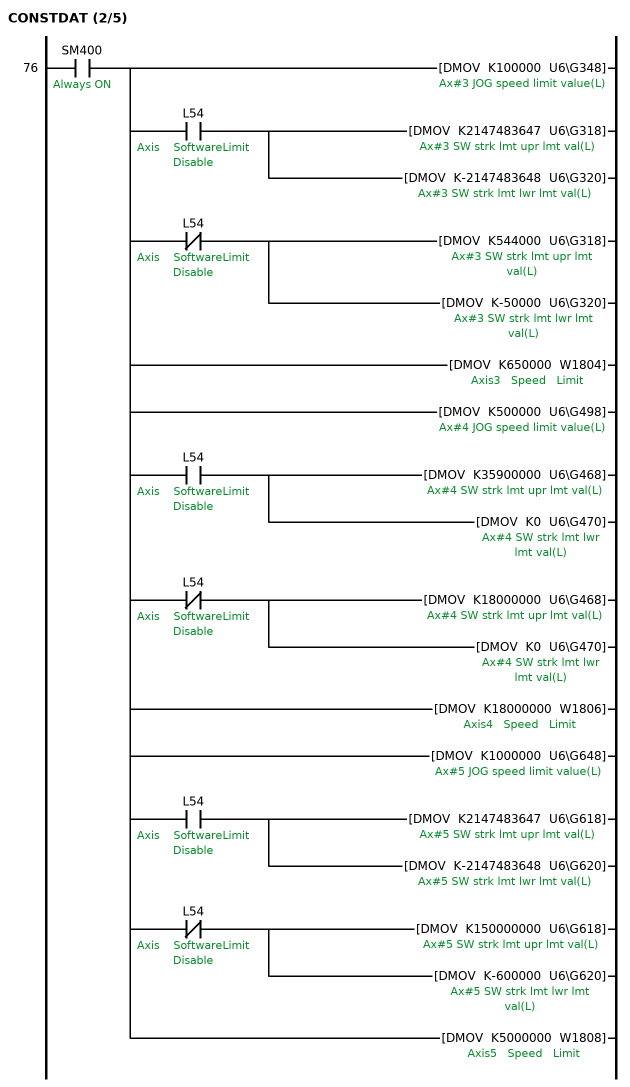
[picture p48: ladder of CONSTDAT, rungs at steps 76 to 76]
76    LD      SM400  ; Always ON
      DMOV    K100000 U6\G348  ; Ax#3 JOG speed limit value(L)
      MPS
      AND     L54  ; Axis    SoftwareLimit   Disable
      DMOV    K2147483647 U6\G318  ; Ax#3 SW strk lmt upr lmt val(L)
      DMOV    K-2147483648 U6\G320  ; Ax#3 SW strk lmt lwr lmt val(L)
      MRD
      ANI     L54  ; Axis    SoftwareLimit   Disable
      DMOV    K544000 U6\G318
      DMOV    K-50000 U6\G320
      MPP
      DMOV    K650000 W1804  ; Axis3   Speed   Limit
      DMOV    K500000 U6\G498  ; Ax#4 JOG speed limit value(L)
      MPS
      AND     L54  ; Axis    SoftwareLimit   Disable
      DMOV    K35900000 U6\G468  ; Ax#4 SW strk lmt upr lmt val(L)
      DMOV    K0 U6\G470  ; Ax#4 SW strk lmt lwr lmt val(L)
      MRD
      ANI     L54  ; Axis    SoftwareLimit   Disable
      DMOV    K18000000 U6\G468
      DMOV    K0 U6\G470
      MPP
      DMOV    K18000000 W1806  ; Axis4   Speed   Limit
      DMOV    K1000000 U6\G648  ; Ax#5 JOG speed limit value(L)
      MPS
      AND     L54  ; Axis    SoftwareLimit   Disable
      DMOV    K2147483647 U6\G618  ; Ax#5 SW strk lmt upr lmt val(L)
      DMOV    K-2147483648 U6\G620  ; Ax#5 SW strk lmt lwr lmt val(L)
      MRD
      ANI     L54  ; Axis    SoftwareLimit   Disable
      DMOV    K150000000 U6\G618
      DMOV    K-600000 U6\G620
      MPP
      DMOV    K5000000 W1808  ; Axis5   Speed   Limit
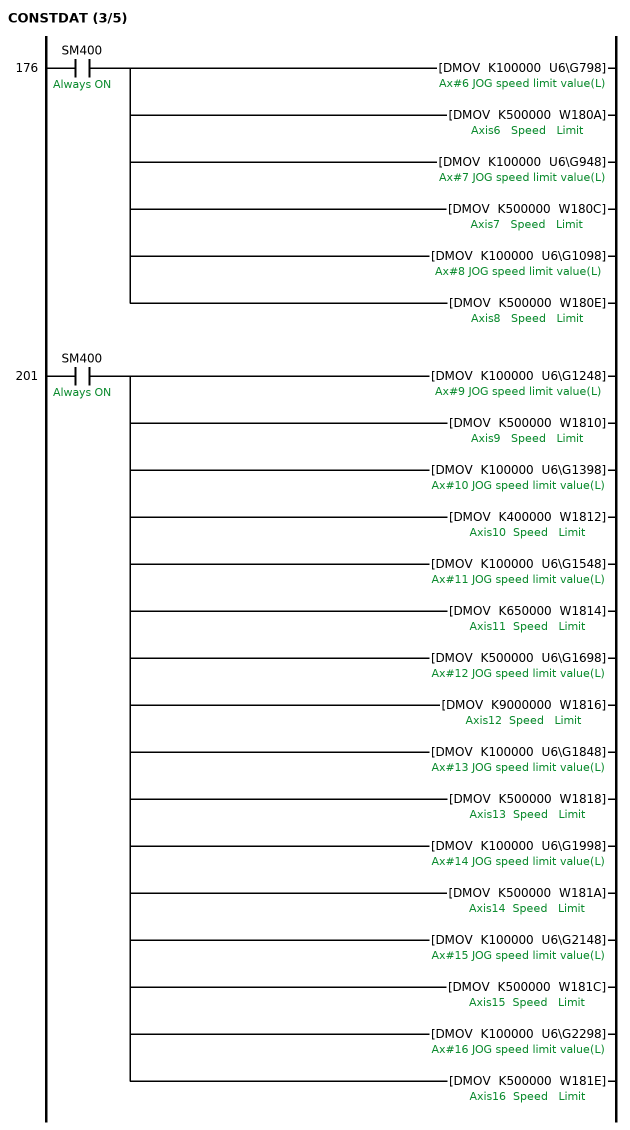
176   LD      SM400  ; Always ON
      DMOV    K100000 U6\G798  ; Ax#6 JOG speed limit value(L)
      DMOV    K500000 W180A  ; Axis6   Speed   Limit
      DMOV    K100000 U6\G948  ; Ax#7 JOG speed limit value(L)
      DMOV    K500000 W180C  ; Axis7   Speed   Limit
      DMOV    K100000 U6\G1098  ; Ax#8 JOG speed limit value(L)
      DMOV    K500000 W180E  ; Axis8   Speed   Limit
201   LD      SM400  ; Always ON
      DMOV    K100000 U6\G1248  ; Ax#9 JOG speed limit value(L)
      DMOV    K500000 W1810  ; Axis9   Speed   Limit
      DMOV    K100000 U6\G1398  ; Ax#10 JOG speed limit value(L)
      DMOV    K400000 W1812  ; Axis10  Speed   Limit
      DMOV    K100000 U6\G1548  ; Ax#11 JOG speed limit value(L)
      DMOV    K650000 W1814  ; Axis11  Speed   Limit
      DMOV    K500000 U6\G1698  ; Ax#12 JOG speed limit value(L)
      DMOV    K9000000 W1816  ; Axis12  Speed   Limit
      DMOV    K100000 U6\G1848  ; Ax#13 JOG speed limit value(L)
      DMOV    K500000 W1818  ; Axis13  Speed   Limit
      DMOV    K100000 U6\G1998  ; Ax#14 JOG speed limit value(L)
      DMOV    K500000 W181A  ; Axis14  Speed   Limit
      DMOV    K100000 U6\G2148  ; Ax#15 JOG speed limit value(L)
      DMOV    K500000 W181C  ; Axis15  Speed   Limit
      DMOV    K100000 U6\G2298  ; Ax#16 JOG speed limit value(L)
      DMOV    K500000 W181E  ; Axis16  Speed   Limit
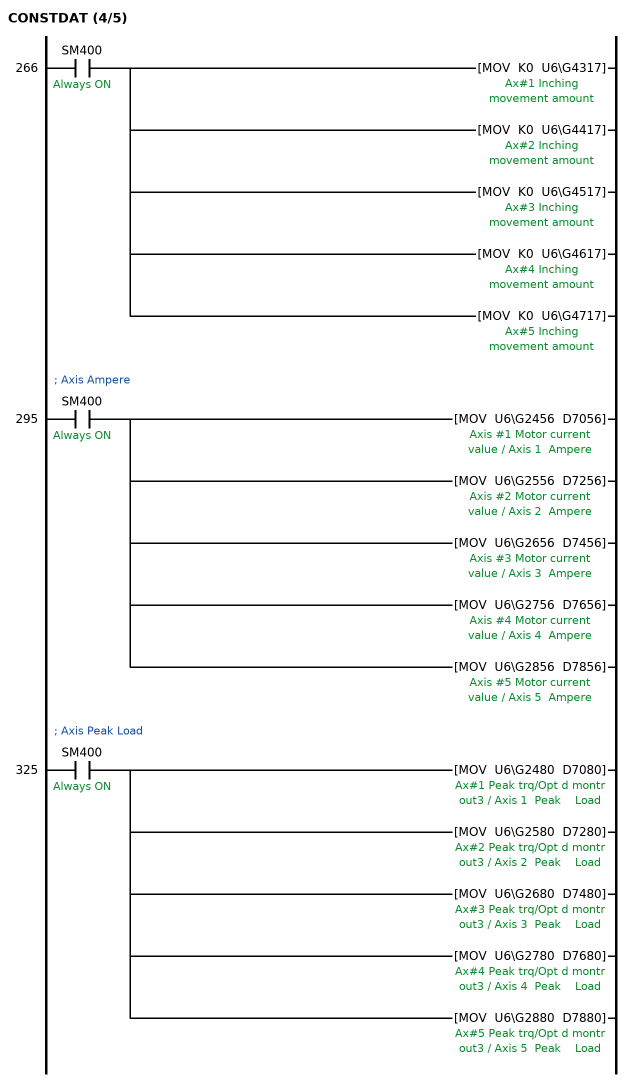
266   LD      SM400  ; Always ON
      MOV     K0 U6\G4317  ; Ax#1 Inching movement amount
      MOV     K0 U6\G4417  ; Ax#2 Inching movement amount
      MOV     K0 U6\G4517  ; Ax#3 Inching movement amount
      MOV     K0 U6\G4617  ; Ax#4 Inching movement amount
      MOV     K0 U6\G4717  ; Ax#5 Inching movement amount
; Axis Ampere
295   LD      SM400  ; Always ON
      MOV     U6\G2456 D7056  ; Axis #1 Motor current value / Axis 1  Ampere
      MOV     U6\G2556 D7256  ; Axis #2 Motor current value / Axis 2  Ampere
      MOV     U6\G2656 D7456  ; Axis #3 Motor current value / Axis 3  Ampere
      MOV     U6\G2756 D7656  ; Axis #4 Motor current value / Axis 4  Ampere
      MOV     U6\G2856 D7856  ; Axis #5 Motor current value / Axis 5  Ampere
; Axis Peak Load
325   LD      SM400  ; Always ON
      MOV     U6\G2480 D7080  ; Ax#1 Peak trq/Opt d montr out3 / Axis 1  Peak    Load
      MOV     U6\G2580 D7280  ; Ax#2 Peak trq/Opt d montr out3 / Axis 2  Peak    Load
      MOV     U6\G2680 D7480  ; Ax#3 Peak trq/Opt d montr out3 / Axis 3  Peak    Load
      MOV     U6\G2780 D7680  ; Ax#4 Peak trq/Opt d montr out3 / Axis 4  Peak    Load
      MOV     U6\G2880 D7880  ; Ax#5 Peak trq/Opt d montr out3 / Axis 5  Peak    Load
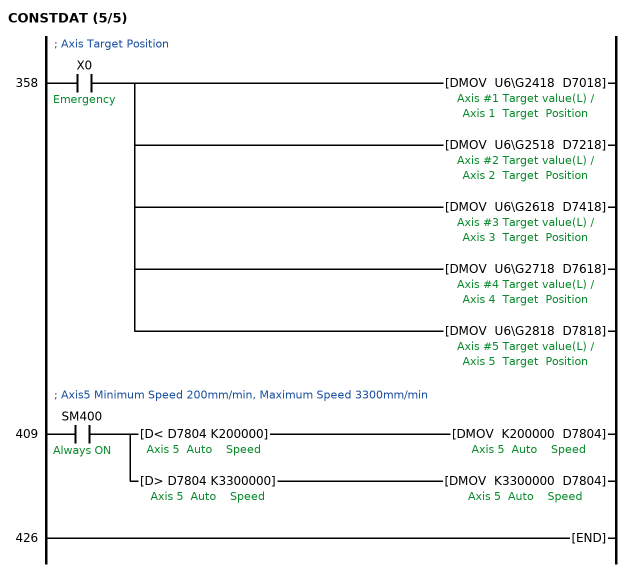
; Axis Target Position
358   LD      X0  ; Emergency
      DMOV    U6\G2418 D7018  ; Axis #1 Target value(L) / Axis 1  Target  Position
      DMOV    U6\G2518 D7218  ; Axis #2 Target value(L) / Axis 2  Target  Position
      DMOV    U6\G2618 D7418  ; Axis #3 Target value(L) / Axis 3  Target  Position
      DMOV    U6\G2718 D7618  ; Axis #4 Target value(L) / Axis 4  Target  Position
      DMOV    U6\G2818 D7818  ; Axis #5 Target value(L) / Axis 5  Target  Position
; Axis5 Minimum Speed 200mm/min, Maximum Speed 3300mm/min
409   LD      SM400  ; Always ON
      MPS
      ANDD<   D7804 K200000  ; Axis 5  Auto    Speed
      DMOV    K200000 D7804
      MPP
      ANDD>   D7804 K3300000  ; Axis 5  Auto    Speed
      DMOV    K3300000 D7804
426   END
END_PROGRAM

PROGRAM Y_OUT
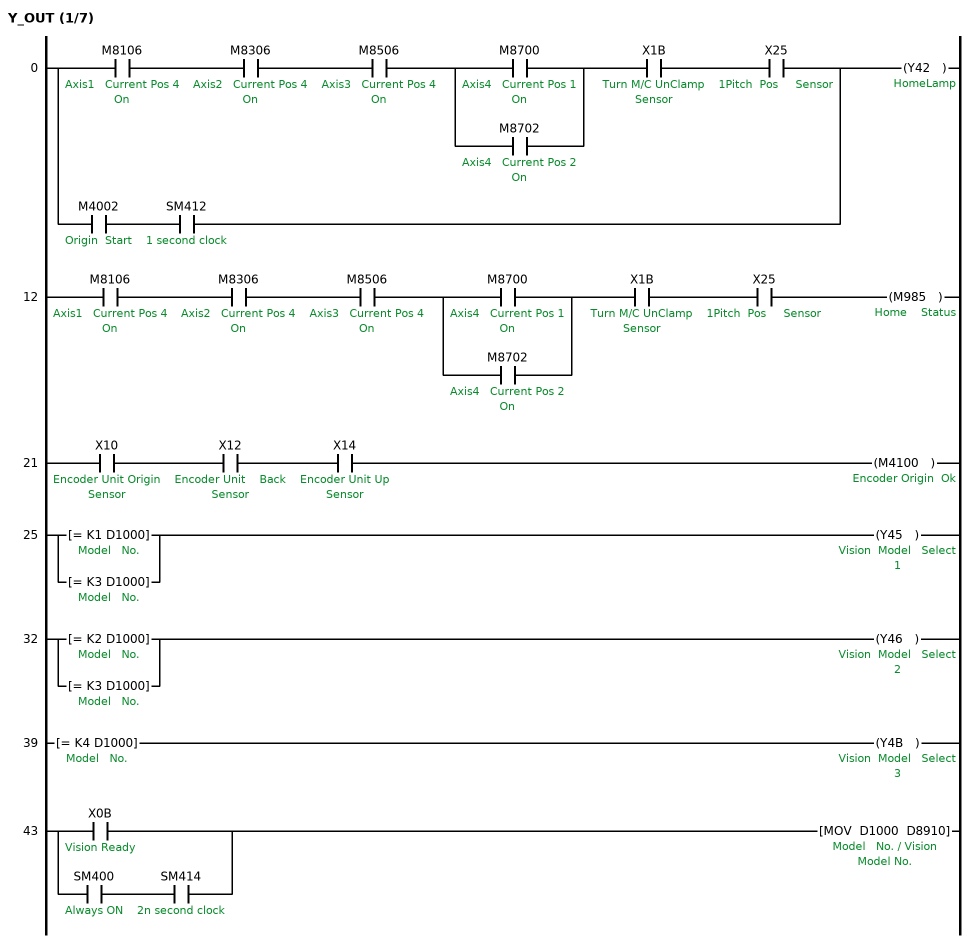
0     LD      M8106  ; Axis1   Current Pos 4 On
      AND     M8306  ; Axis2   Current Pos 4 On
      AND     M8506  ; Axis3   Current Pos 4 On
      LD      M8700  ; Axis4   Current Pos 1 On
      OR      M8702  ; Axis4   Current Pos 2 On
      ANB
      AND     X1B  ; Turn M/C UnClamp Sensor
      AND     X25  ; 1Pitch  Pos     Sensor
      LD      M4002  ; Origin  Start
      AND     SM412  ; 1 second clock
      ORB
      OUT     Y42  ; HomeLamp
12    LD      M8106  ; Axis1   Current Pos 4 On
      AND     M8306  ; Axis2   Current Pos 4 On
      AND     M8506  ; Axis3   Current Pos 4 On
      LD      M8700  ; Axis4   Current Pos 1 On
      OR      M8702  ; Axis4   Current Pos 2 On
      ANB
      AND     X1B  ; Turn M/C UnClamp Sensor
      AND     X25  ; 1Pitch  Pos     Sensor
      OUT     M985  ; Home    Status
21    LD      X10  ; Encoder Unit Origin Sensor
      AND     X12  ; Encoder Unit    Back    Sensor
      AND     X14  ; Encoder Unit Up Sensor
      OUT     M4100  ; Encoder Origin  Ok
25    LD=     K1 D1000  ; Model   No.
      OR=     K3 D1000  ; Model   No.
      OUT     Y45  ; Vision  Model   Select 1
32    LD=     K2 D1000  ; Model   No.
      OR=     K3 D1000  ; Model   No.
      OUT     Y46  ; Vision  Model   Select 2
39    LD=     K4 D1000  ; Model   No.
      OUT     Y4B  ; Vision  Model   Select 3
43    LD      X0B  ; Vision Ready
      LD      SM400  ; Always ON
      AND     SM414  ; 2n second clock
      ORB
      MOV     D1000 D8910  ; Vision Model No.
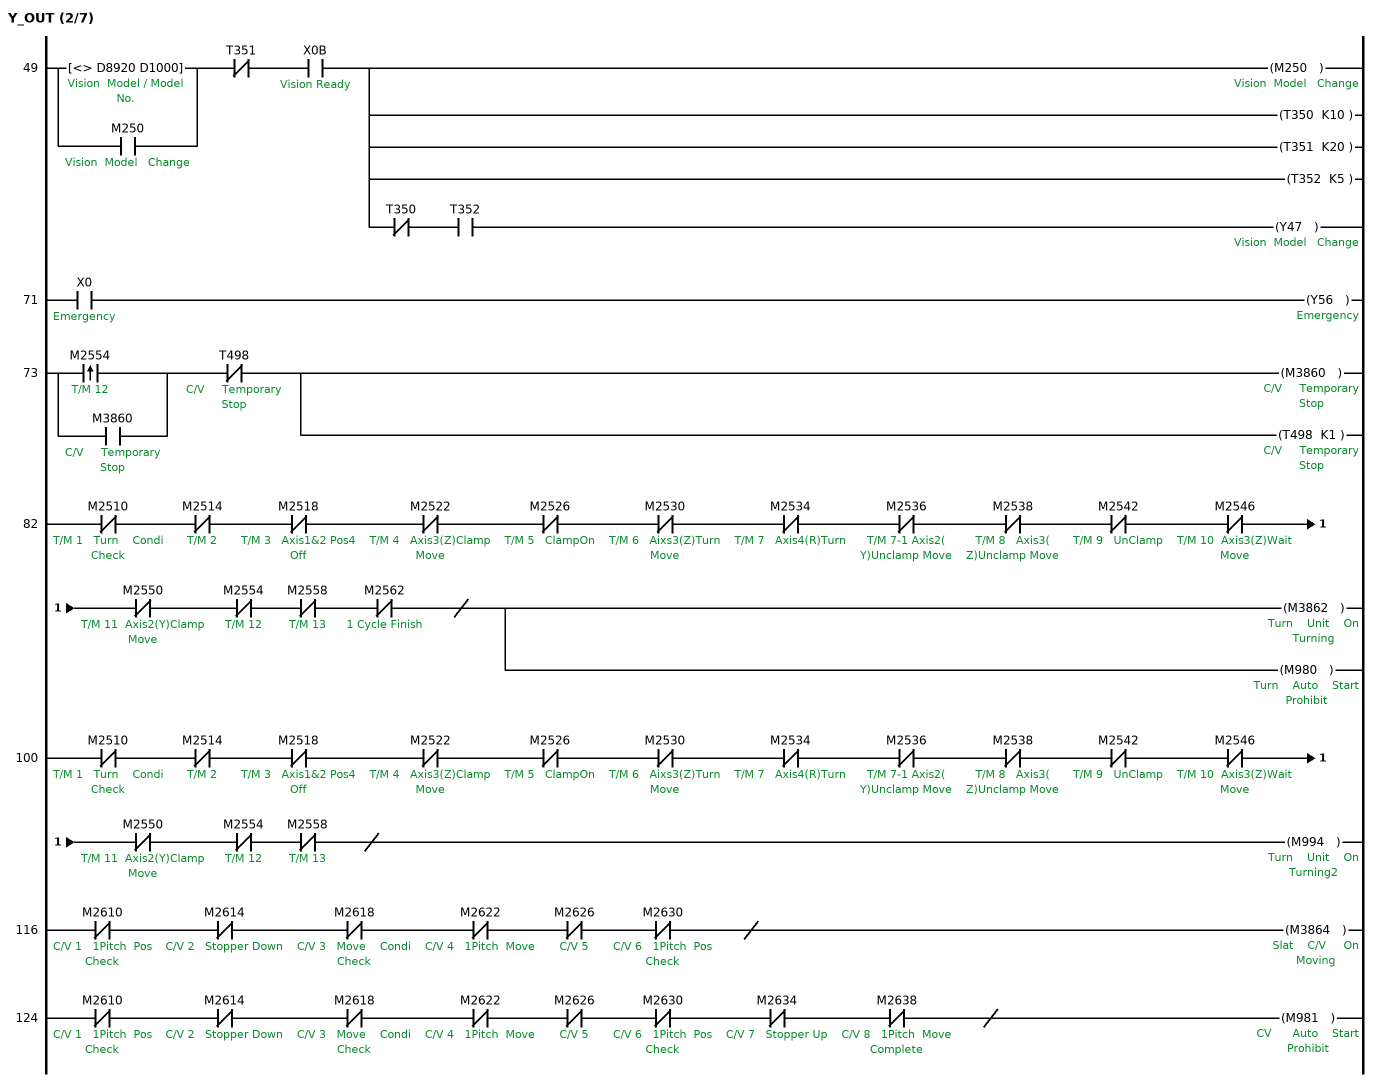
49    LD<>    D8920 D1000  ; Vision  Model / Model   No.
      OR      M250  ; Vision  Model   Change
      ANI     T351
      AND     X0B  ; Vision Ready
      OUT     M250  ; Vision  Model   Change
      OUT     T350 K10
      OUT     T351 K20
      OUT     T352 K5
      ANI     T350
      AND     T352
      OUT     Y47  ; Vision  Model   Change
71    LD      X0  ; Emergency
      OUT     Y56  ; Emergency
73    LDP     M2554  ; T/M 12
      OR      M3860  ; C/V     Temporary  Stop
      ANI     T498  ; C/V     Temporary  Stop
      OUT     M3860  ; C/V     Temporary  Stop
      OUT     T498 K1  ; C/V     Temporary  Stop
82    LDI     M2510  ; T/M 1   Turn    Condi   Check
      ANI     M2514  ; T/M 2
      ANI     M2518  ; T/M 3   Axis1&2 Pos4    Off
      ANI     M2522  ; T/M 4   Axis3(Z)Clamp   Move
      ANI     M2526  ; T/M 5   ClampOn
      ANI     M2530  ; T/M 6   Aixs3(Z)Turn    Move
      ANI     M2534  ; T/M 7   Axis4(R)Turn
      ANI     M2536  ; T/M 7-1 Axis2(Y)Unclamp Move
      ANI     M2538  ; T/M 8   Axis3(Z)Unclamp Move
      ANI     M2542  ; T/M 9   UnClamp
      ANI     M2546  ; T/M 10  Axis3(Z)Wait    Move
      ANI     M2550  ; T/M 11  Axis2(Y)Clamp   Move
      ANI     M2554  ; T/M 12
      ANI     M2558  ; T/M 13
      ANI     M2562  ; 1 Cycle Finish
      INV
      OUT     M3862  ; Turn    Unit    On      Turning
      OUT     M980  ; Turn    Auto    Start   Prohibit
100   LDI     M2510  ; T/M 1   Turn    Condi   Check
      ANI     M2514  ; T/M 2
      ANI     M2518  ; T/M 3   Axis1&2 Pos4    Off
      ANI     M2522  ; T/M 4   Axis3(Z)Clamp   Move
      ANI     M2526  ; T/M 5   ClampOn
      ANI     M2530  ; T/M 6   Aixs3(Z)Turn    Move
      ANI     M2534  ; T/M 7   Axis4(R)Turn
      ANI     M2536  ; T/M 7-1 Axis2(Y)Unclamp Move
      ANI     M2538  ; T/M 8   Axis3(Z)Unclamp Move
      ANI     M2542  ; T/M 9   UnClamp
      ANI     M2546  ; T/M 10  Axis3(Z)Wait    Move
      ANI     M2550  ; T/M 11  Axis2(Y)Clamp   Move
      ANI     M2554  ; T/M 12
      ANI     M2558  ; T/M 13
      INV
      OUT     M994  ; Turn    Unit    On      Turning2
116   LDI     M2610  ; C/V 1   1Pitch  Pos     Check
      ANI     M2614  ; C/V 2   Stopper Down
      ANI     M2618  ; C/V 3   Move    Condi   Check
      ANI     M2622  ; C/V 4   1Pitch  Move
      ANI     M2626  ; C/V 5
      ANI     M2630  ; C/V 6   1Pitch  Pos     Check
      INV
      OUT     M3864  ; Slat    C/V     On      Moving
124   LDI     M2610  ; C/V 1   1Pitch  Pos     Check
      ANI     M2614  ; C/V 2   Stopper Down
      ANI     M2618  ; C/V 3   Move    Condi   Check
      ANI     M2622  ; C/V 4   1Pitch  Move
      ANI     M2626  ; C/V 5
      ANI     M2630  ; C/V 6   1Pitch  Pos     Check
      ANI     M2634  ; C/V 7   Stopper Up
      ANI     M2638  ; C/V 8   1Pitch  Move    Complete
      INV
      OUT     M981  ; CV      Auto    Start   Prohibit
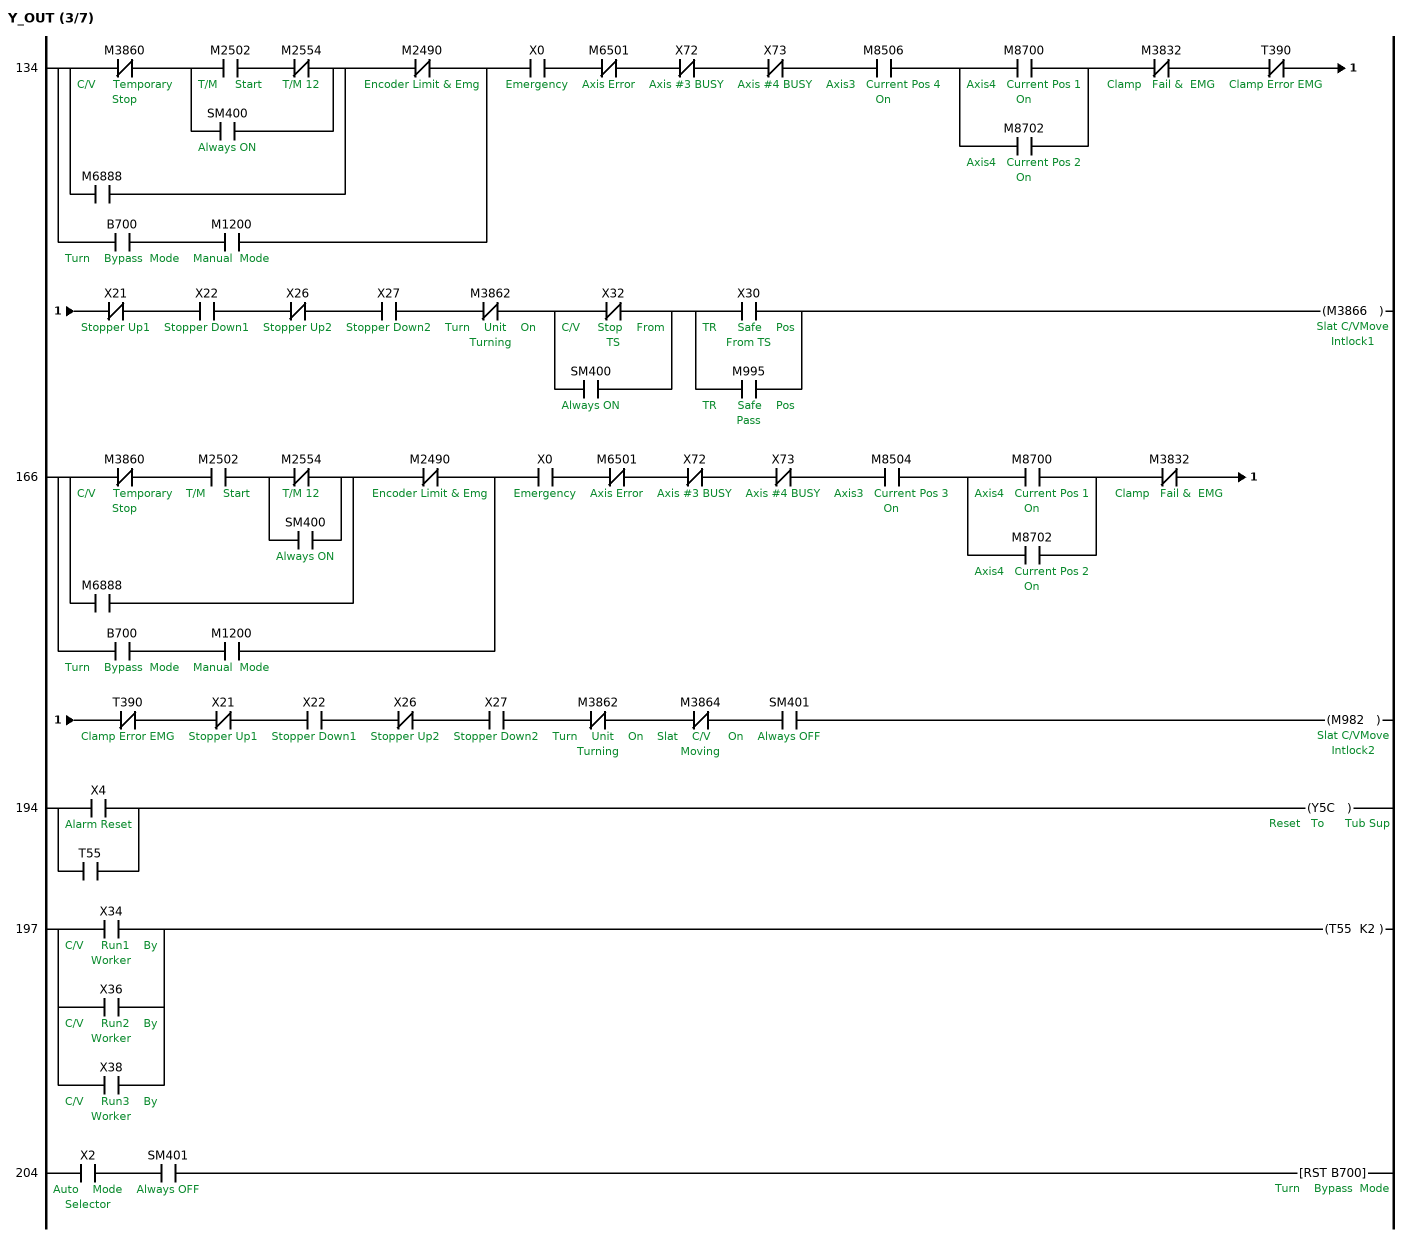
134   LDI     M3860  ; C/V     Temporary  Stop
      LD      M2502  ; T/M     Start
      ANI     M2554  ; T/M 12
      OR      SM400  ; Always ON
      ANB
      OR      M6888
      ANI     M2490  ; Encoder Limit & Emg
      LD      B700  ; Turn    Bypass  Mode
      AND     M1200  ; Manual  Mode
      ORB
      AND     X0  ; Emergency
      ANI     M6501  ; Axis Error
      ANI     X72  ; Axis #3 BUSY
      ANI     X73  ; Axis #4 BUSY
      AND     M8506  ; Axis3   Current Pos 4 On
      LD      M8700  ; Axis4   Current Pos 1 On
      OR      M8702  ; Axis4   Current Pos 2 On
      ANB
      ANI     M3832  ; Clamp   Fail &  EMG
      ANI     T390  ; Clamp Error EMG
      ANI     X21  ; Stopper Up1
      AND     X22  ; Stopper Down1
      ANI     X26  ; Stopper Up2
      AND     X27  ; Stopper Down2
      ANI     M3862  ; Turn    Unit    On      Turning
      LDI     X32  ; C/V     Stop    From    TS
      OR      SM400  ; Always ON
      ANB
      LD      X30  ; TR      Safe    Pos     From TS
      OR      M995  ; TR      Safe    Pos     Pass
      ANB
      OUT     M3866  ; Slat C/VMove    Intlock1
166   LDI     M3860  ; C/V     Temporary  Stop
      AND     M2502  ; T/M     Start
      LDI     M2554  ; T/M 12
      OR      SM400  ; Always ON
      ANB
      OR      M6888
      ANI     M2490  ; Encoder Limit & Emg
      LD      B700  ; Turn    Bypass  Mode
      AND     M1200  ; Manual  Mode
      ORB
      AND     X0  ; Emergency
      ANI     M6501  ; Axis Error
      ANI     X72  ; Axis #3 BUSY
      ANI     X73  ; Axis #4 BUSY
      AND     M8504  ; Axis3   Current Pos 3 On
      LD      M8700  ; Axis4   Current Pos 1 On
      OR      M8702  ; Axis4   Current Pos 2 On
      ANB
      ANI     M3832  ; Clamp   Fail &  EMG
      ANI     T390  ; Clamp Error EMG
      ANI     X21  ; Stopper Up1
      AND     X22  ; Stopper Down1
      ANI     X26  ; Stopper Up2
      AND     X27  ; Stopper Down2
      ANI     M3862  ; Turn    Unit    On      Turning
      ANI     M3864  ; Slat    C/V     On      Moving
      AND     SM401  ; Always OFF
      OUT     M982  ; Slat C/VMove    Intlock2
194   LD      X4  ; Alarm Reset
      OR      T55
      OUT     Y5C  ; Reset   To      Tub Sup
197   LD      X34  ; C/V     Run1    By      Worker
      OR      X36  ; C/V     Run2    By      Worker
      OR      X38  ; C/V     Run3    By      Worker
      OUT     T55 K2
204   LD      X2  ; Auto    Mode    Selector
      AND     SM401  ; Always OFF
      RST     B700  ; Turn    Bypass  Mode
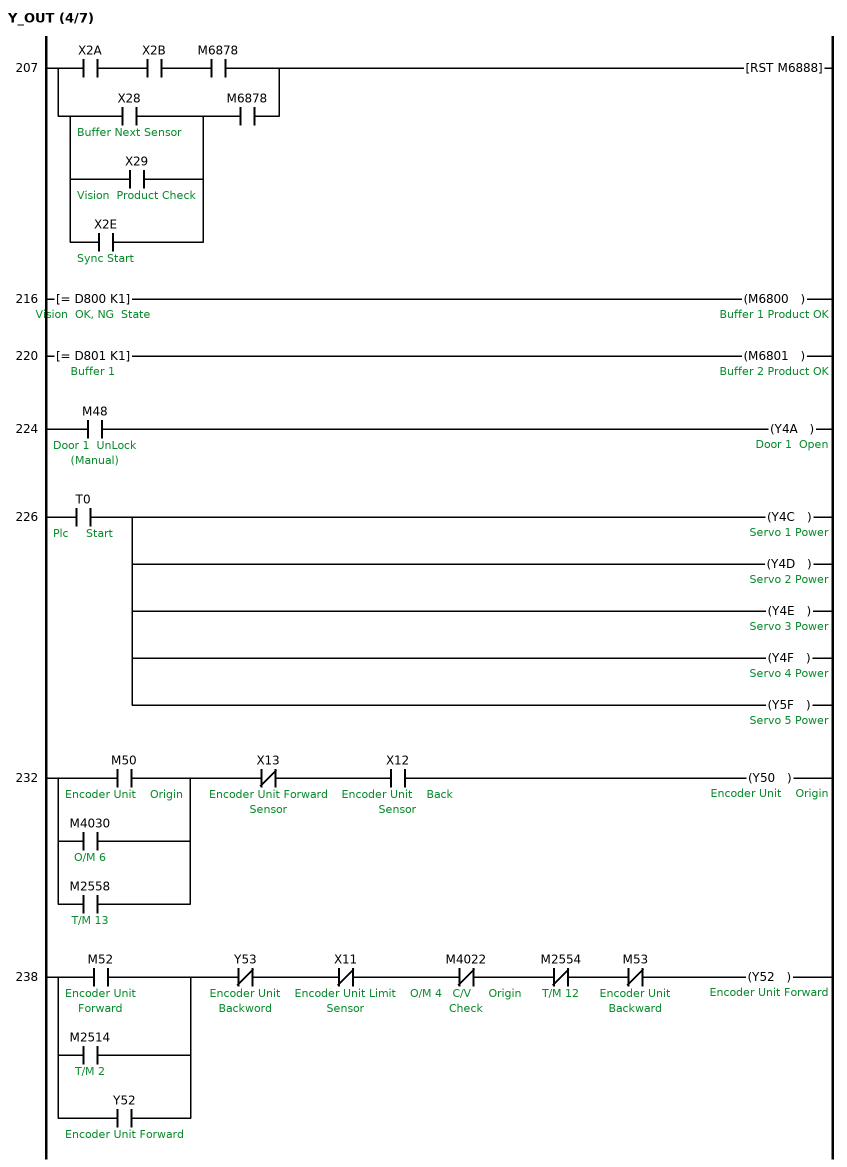
207   LD      X2A
      AND     X2B
      AND     M6878
      LD      X28  ; Buffer Next Sensor
      OR      X29  ; Vision  Product Check
      OR      X2E  ; Sync Start
      AND     M6878
      ORB
      RST     M6888
216   LD=     D800 K1  ; Vision  OK, NG  State
      OUT     M6800  ; Buffer 1 Product OK
220   LD=     D801 K1  ; Buffer 1
      OUT     M6801  ; Buffer 2 Product OK
224   LD      M48  ; Door 1  UnLock  (Manual)
      OUT     Y4A  ; Door 1  Open
226   LD      T0  ; Plc     Start
      OUT     Y4C  ; Servo 1 Power
      OUT     Y4D  ; Servo 2 Power
      OUT     Y4E  ; Servo 3 Power
      OUT     Y4F  ; Servo 4 Power
      OUT     Y5F  ; Servo 5 Power
232   LD      M50  ; Encoder Unit    Origin
      OR      M4030  ; O/M 6
      OR      M2558  ; T/M 13
      ANI     X13  ; Encoder Unit Forward Sensor
      AND     X12  ; Encoder Unit    Back    Sensor
      OUT     Y50  ; Encoder Unit    Origin
238   LD      M52  ; Encoder Unit    Forward
      OR      M2514  ; T/M 2
      OR      Y52  ; Encoder Unit Forward
      ANI     Y53  ; Encoder Unit Backword
      ANI     X11  ; Encoder Unit Limit Sensor
      ANI     M4022  ; O/M 4   C/V     Origin  Check
      ANI     M2554  ; T/M 12
      ANI     M53  ; Encoder Unit    Backward
      OUT     Y52  ; Encoder Unit Forward
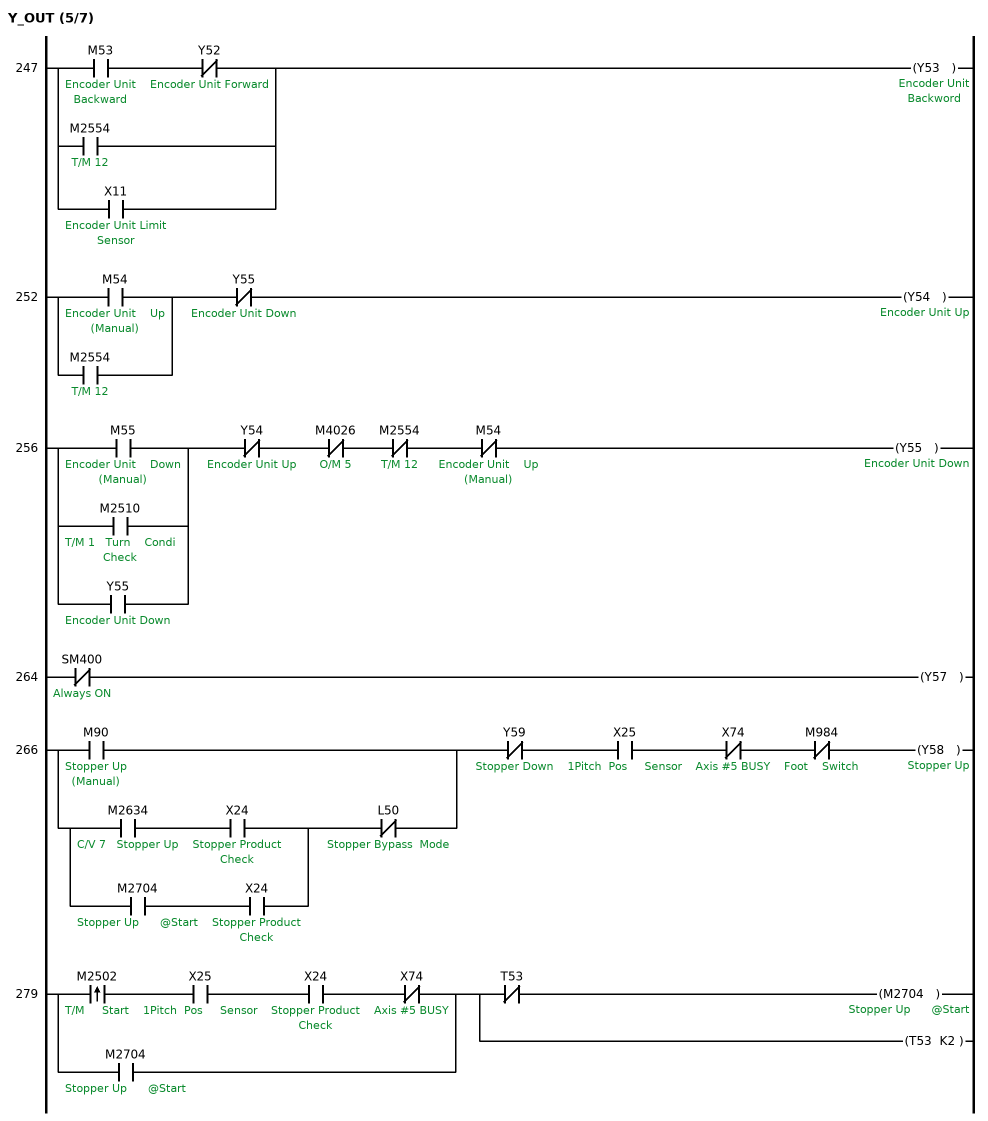
247   LD      M53  ; Encoder Unit    Backward
      ANI     Y52  ; Encoder Unit Forward
      OR      M2554  ; T/M 12
      OR      X11  ; Encoder Unit Limit Sensor
      OUT     Y53  ; Encoder Unit Backword
252   LD      M54  ; Encoder Unit    Up      (Manual)
      OR      M2554  ; T/M 12
      ANI     Y55  ; Encoder Unit Down
      OUT     Y54  ; Encoder Unit Up
256   LD      M55  ; Encoder Unit    Down    (Manual)
      OR      M2510  ; T/M 1   Turn    Condi   Check
      OR      Y55  ; Encoder Unit Down
      ANI     Y54  ; Encoder Unit Up
      ANI     M4026  ; O/M 5
      ANI     M2554  ; T/M 12
      ANI     M54  ; Encoder Unit    Up      (Manual)
      OUT     Y55  ; Encoder Unit Down
264   LDI     SM400  ; Always ON
      OUT     Y57
266   LD      M90  ; Stopper Up      (Manual)
      LD      M2634  ; C/V 7   Stopper Up
      AND     X24  ; Stopper Product Check
      LD      M2704  ; Stopper Up      @Start
      AND     X24  ; Stopper Product Check
      ORB
      ANI     L50  ; Stopper Bypass  Mode
      ORB
      ANI     Y59  ; Stopper Down
      AND     X25  ; 1Pitch  Pos     Sensor
      ANI     X74  ; Axis #5 BUSY
      ANI     M984  ; Foot    Switch
      OUT     Y58  ; Stopper Up
279   LDP     M2502  ; T/M     Start
      AND     X25  ; 1Pitch  Pos     Sensor
      AND     X24  ; Stopper Product Check
      ANI     X74  ; Axis #5 BUSY
      OR      M2704  ; Stopper Up      @Start
      MPS
      ANI     T53
      OUT     M2704  ; Stopper Up      @Start
      MPP
      OUT     T53 K2
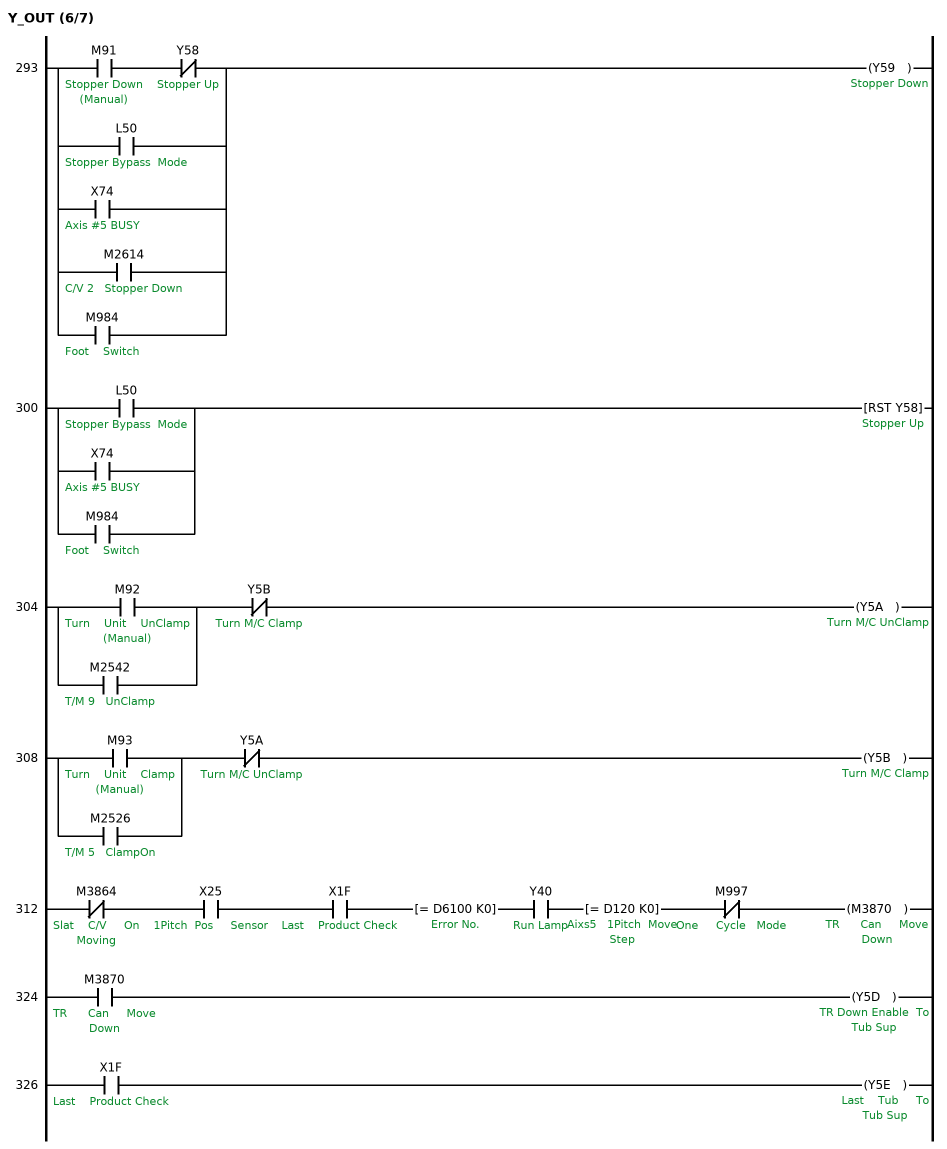
293   LD      M91  ; Stopper Down    (Manual)
      ANI     Y58  ; Stopper Up
      OR      L50  ; Stopper Bypass  Mode
      OR      X74  ; Axis #5 BUSY
      OR      M2614  ; C/V 2   Stopper Down
      OR      M984  ; Foot    Switch
      OUT     Y59  ; Stopper Down
300   LD      L50  ; Stopper Bypass  Mode
      OR      X74  ; Axis #5 BUSY
      OR      M984  ; Foot    Switch
      RST     Y58  ; Stopper Up
304   LD      M92  ; Turn    Unit    UnClamp (Manual)
      OR      M2542  ; T/M 9   UnClamp
      ANI     Y5B  ; Turn M/C Clamp
      OUT     Y5A  ; Turn M/C UnClamp
308   LD      M93  ; Turn    Unit    Clamp   (Manual)
      OR      M2526  ; T/M 5   ClampOn
      ANI     Y5A  ; Turn M/C UnClamp
      OUT     Y5B  ; Turn M/C Clamp
312   LDI     M3864  ; Slat    C/V     On      Moving
      AND     X25  ; 1Pitch  Pos     Sensor
      AND     X1F  ; Last    Product Check
      AND=    D6100 K0  ; Error No.
      AND     Y40  ; Run Lamp
      AND=    D120 K0  ; Aixs5   1Pitch  Move    Step
      ANI     M997  ; One     Cycle   Mode
      OUT     M3870  ; TR      Can     Move    Down
324   LD      M3870  ; TR      Can     Move    Down
      OUT     Y5D  ; TR Down Enable  To      Tub Sup
326   LD      X1F  ; Last    Product Check
      OUT     Y5E  ; Last    Tub     To      Tub Sup
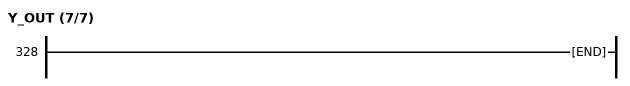
328   END
END_PROGRAM

PROGRAM POS_DATA
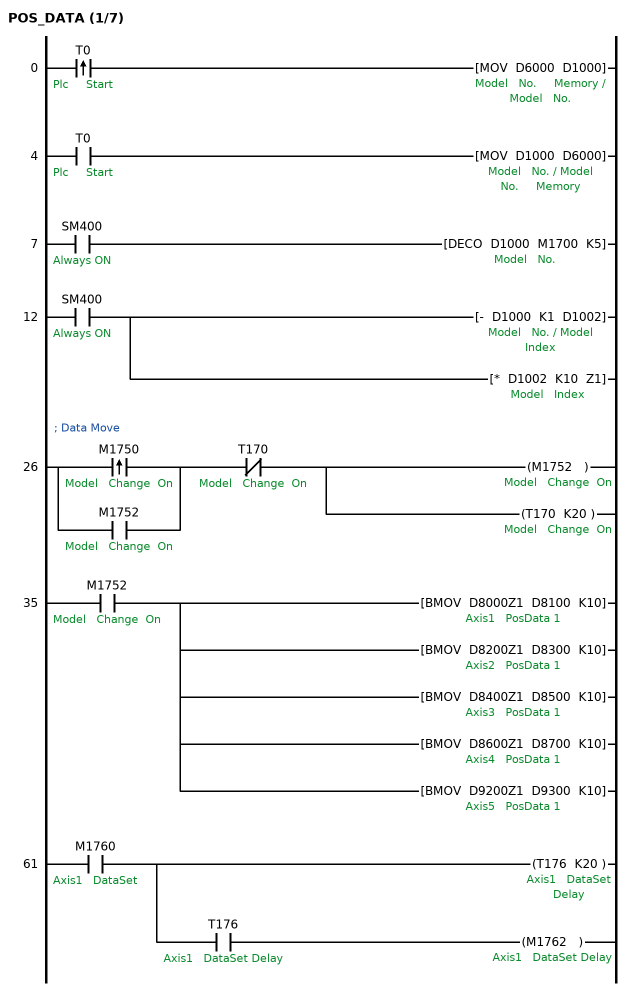
0     LDP     T0  ; Plc     Start
      MOV     D6000 D1000  ; Model   No.     Memory / Model   No.
4     LD      T0  ; Plc     Start
      MOV     D1000 D6000
7     LD      SM400  ; Always ON
      DECO    D1000 M1700 K5
12    LD      SM400  ; Always ON
      -       D1000 K1 D1002  ; Model   Index
      *       D1002 K10 Z1
; Data Move
26    LDP     M1750  ; Model   Change  On
      OR      M1752  ; Model   Change  On
      ANI     T170  ; Model   Change  On
      OUT     M1752  ; Model   Change  On
      OUT     T170 K20  ; Model   Change  On
35    LD      M1752  ; Model   Change  On
      BMOV    D8000Z1 D8100 K10  ; Axis1   PosData 1
      BMOV    D8200Z1 D8300 K10  ; Axis2   PosData 1
      BMOV    D8400Z1 D8500 K10  ; Axis3   PosData 1
      BMOV    D8600Z1 D8700 K10  ; Axis4   PosData 1
      BMOV    D9200Z1 D9300 K10  ; Axis5   PosData 1
61    LD      M1760  ; Axis1   DataSet
      OUT     T176 K20  ; Axis1   DataSet Delay
      AND     T176  ; Axis1   DataSet Delay
      OUT     M1762  ; Axis1   DataSet Delay
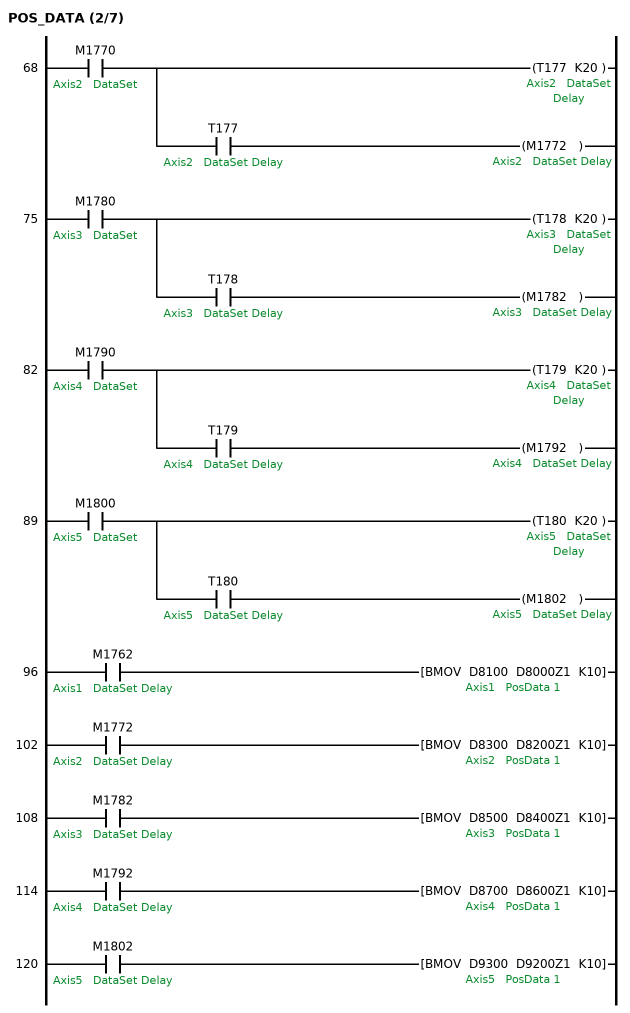
68    LD      M1770  ; Axis2   DataSet
      OUT     T177 K20  ; Axis2   DataSet Delay
      AND     T177  ; Axis2   DataSet Delay
      OUT     M1772  ; Axis2   DataSet Delay
75    LD      M1780  ; Axis3   DataSet
      OUT     T178 K20  ; Axis3   DataSet Delay
      AND     T178  ; Axis3   DataSet Delay
      OUT     M1782  ; Axis3   DataSet Delay
82    LD      M1790  ; Axis4   DataSet
      OUT     T179 K20  ; Axis4   DataSet Delay
      AND     T179  ; Axis4   DataSet Delay
      OUT     M1792  ; Axis4   DataSet Delay
89    LD      M1800  ; Axis5   DataSet
      OUT     T180 K20  ; Axis5   DataSet Delay
      AND     T180  ; Axis5   DataSet Delay
      OUT     M1802  ; Axis5   DataSet Delay
96    LD      M1762  ; Axis1   DataSet Delay
      BMOV    D8100 D8000Z1 K10
102   LD      M1772  ; Axis2   DataSet Delay
      BMOV    D8300 D8200Z1 K10
108   LD      M1782  ; Axis3   DataSet Delay
      BMOV    D8500 D8400Z1 K10
114   LD      M1792  ; Axis4   DataSet Delay
      BMOV    D8700 D8600Z1 K10
120   LD      M1802  ; Axis5   DataSet Delay
      BMOV    D9300 D9200Z1 K10
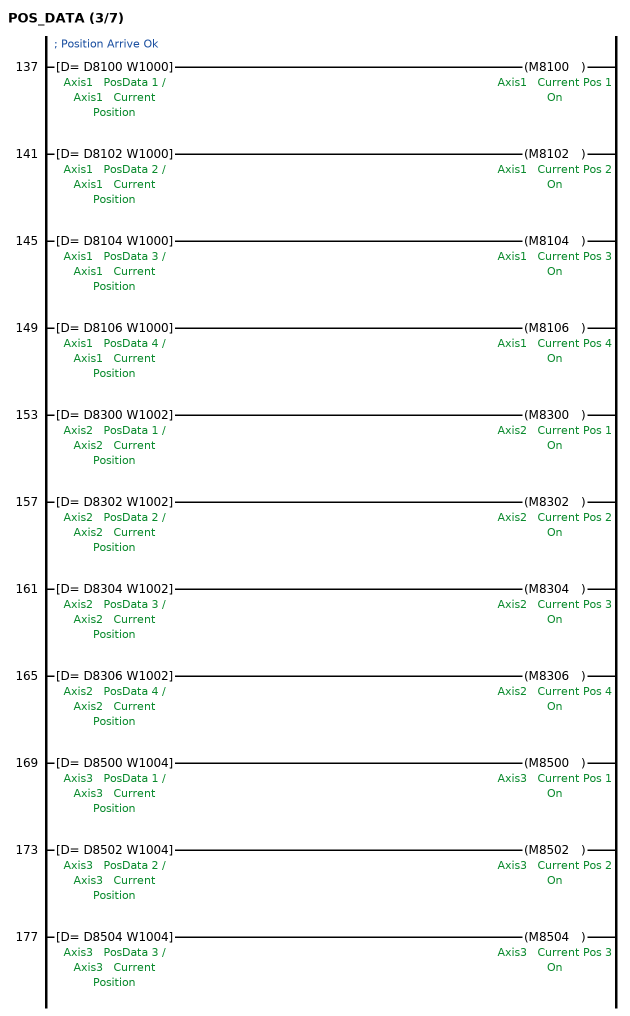
; Position Arrive Ok
137   LDD=    D8100 W1000  ; Axis1   PosData 1 / Axis1   Current Position
      OUT     M8100  ; Axis1   Current Pos 1 On
141   LDD=    D8102 W1000  ; Axis1   PosData 2 / Axis1   Current Position
      OUT     M8102  ; Axis1   Current Pos 2 On
145   LDD=    D8104 W1000  ; Axis1   PosData 3 / Axis1   Current Position
      OUT     M8104  ; Axis1   Current Pos 3 On
149   LDD=    D8106 W1000  ; Axis1   PosData 4 / Axis1   Current Position
      OUT     M8106  ; Axis1   Current Pos 4 On
153   LDD=    D8300 W1002  ; Axis2   PosData 1 / Axis2   Current Position
      OUT     M8300  ; Axis2   Current Pos 1 On
157   LDD=    D8302 W1002  ; Axis2   PosData 2 / Axis2   Current Position
      OUT     M8302  ; Axis2   Current Pos 2 On
161   LDD=    D8304 W1002  ; Axis2   PosData 3 / Axis2   Current Position
      OUT     M8304  ; Axis2   Current Pos 3 On
165   LDD=    D8306 W1002  ; Axis2   PosData 4 / Axis2   Current Position
      OUT     M8306  ; Axis2   Current Pos 4 On
169   LDD=    D8500 W1004  ; Axis3   PosData 1 / Axis3   Current Position
      OUT     M8500  ; Axis3   Current Pos 1 On
173   LDD=    D8502 W1004  ; Axis3   PosData 2 / Axis3   Current Position
      OUT     M8502  ; Axis3   Current Pos 2 On
177   LDD=    D8504 W1004  ; Axis3   PosData 3 / Axis3   Current Position
      OUT     M8504  ; Axis3   Current Pos 3 On
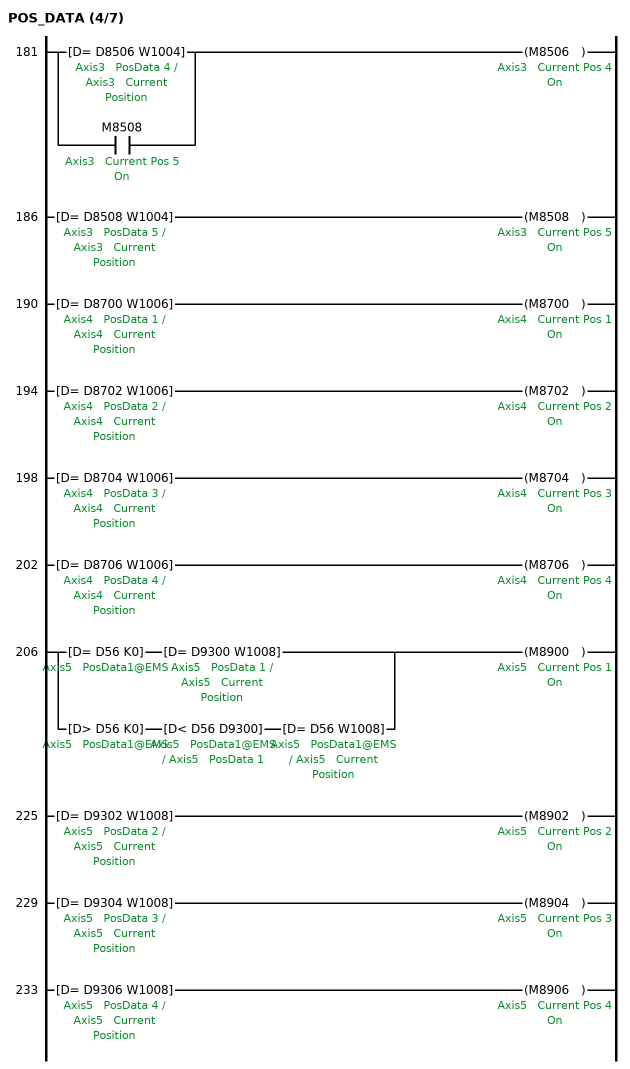
181   LDD=    D8506 W1004  ; Axis3   PosData 4 / Axis3   Current Position
      OR      M8508  ; Axis3   Current Pos 5 On
      OUT     M8506  ; Axis3   Current Pos 4 On
186   LDD=    D8508 W1004  ; Axis3   PosData 5 / Axis3   Current Position
      OUT     M8508  ; Axis3   Current Pos 5 On
190   LDD=    D8700 W1006  ; Axis4   PosData 1 / Axis4   Current Position
      OUT     M8700  ; Axis4   Current Pos 1 On
194   LDD=    D8702 W1006  ; Axis4   PosData 2 / Axis4   Current Position
      OUT     M8702  ; Axis4   Current Pos 2 On
198   LDD=    D8704 W1006  ; Axis4   PosData 3 / Axis4   Current Position
      OUT     M8704  ; Axis4   Current Pos 3 On
202   LDD=    D8706 W1006  ; Axis4   PosData 4 / Axis4   Current Position
      OUT     M8706  ; Axis4   Current Pos 4 On
206   LDD=    D56 K0  ; Axis5   PosData1@EMS
      ANDD=   D9300 W1008  ; Axis5   PosData 1 / Axis5   Current Position
      LDD>    D56 K0  ; Axis5   PosData1@EMS
      ANDD<   D56 D9300  ; Axis5   PosData1@EMS / Axis5   PosData 1
      ANDD=   D56 W1008  ; Axis5   PosData1@EMS / Axis5   Current Position
      ORB
      OUT     M8900  ; Axis5   Current Pos 1 On
225   LDD=    D9302 W1008  ; Axis5   PosData 2 / Axis5   Current Position
      OUT     M8902  ; Axis5   Current Pos 2 On
229   LDD=    D9304 W1008  ; Axis5   PosData 3 / Axis5   Current Position
      OUT     M8904  ; Axis5   Current Pos 3 On
233   LDD=    D9306 W1008  ; Axis5   PosData 4 / Axis5   Current Position
      OUT     M8906  ; Axis5   Current Pos 4 On
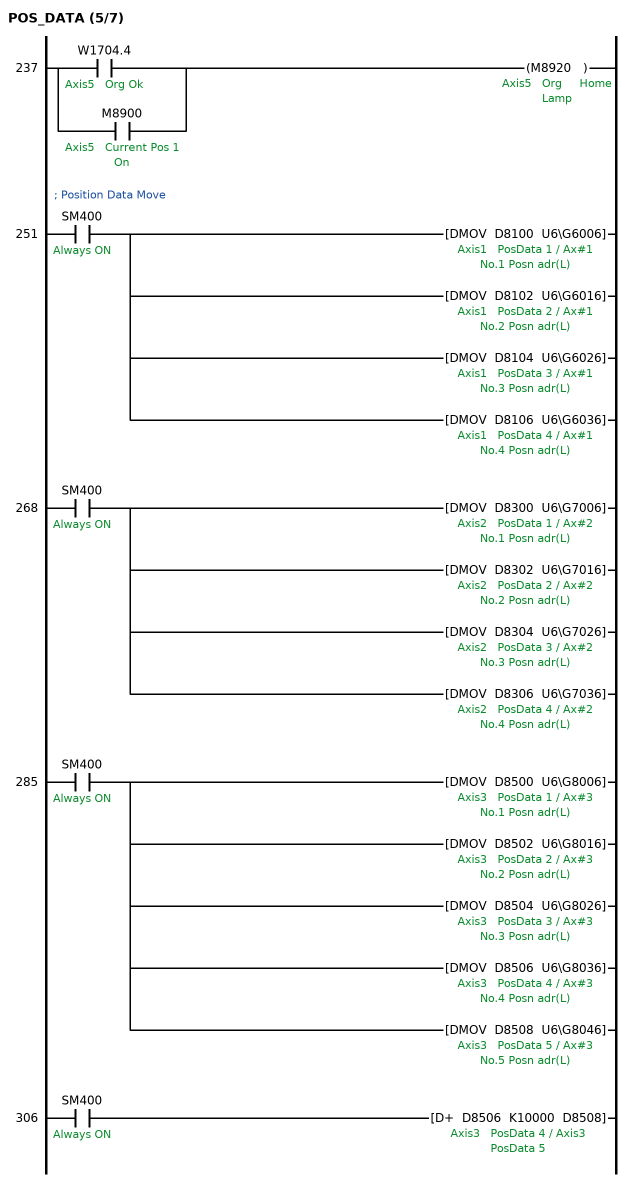
237   LD      W1704.4  ; Axis5   Org Ok
      OR      M8900  ; Axis5   Current Pos 1 On
      OUT     M8920  ; Axis5   Org     Home    Lamp
; Position Data Move
251   LD      SM400  ; Always ON
      DMOV    D8100 U6\G6006  ; Ax#1 No.1 Posn adr(L)
      DMOV    D8102 U6\G6016  ; Ax#1 No.2 Posn adr(L)
      DMOV    D8104 U6\G6026  ; Ax#1 No.3 Posn adr(L)
      DMOV    D8106 U6\G6036  ; Ax#1 No.4 Posn adr(L)
268   LD      SM400  ; Always ON
      DMOV    D8300 U6\G7006  ; Ax#2 No.1 Posn adr(L)
      DMOV    D8302 U6\G7016  ; Ax#2 No.2 Posn adr(L)
      DMOV    D8304 U6\G7026  ; Ax#2 No.3 Posn adr(L)
      DMOV    D8306 U6\G7036  ; Ax#2 No.4 Posn adr(L)
285   LD      SM400  ; Always ON
      DMOV    D8500 U6\G8006  ; Ax#3 No.1 Posn adr(L)
      DMOV    D8502 U6\G8016  ; Ax#3 No.2 Posn adr(L)
      DMOV    D8504 U6\G8026  ; Ax#3 No.3 Posn adr(L)
      DMOV    D8506 U6\G8036  ; Ax#3 No.4 Posn adr(L)
      DMOV    D8508 U6\G8046  ; Ax#3 No.5 Posn adr(L)
306   LD      SM400  ; Always ON
      D+      D8506 K10000 D8508
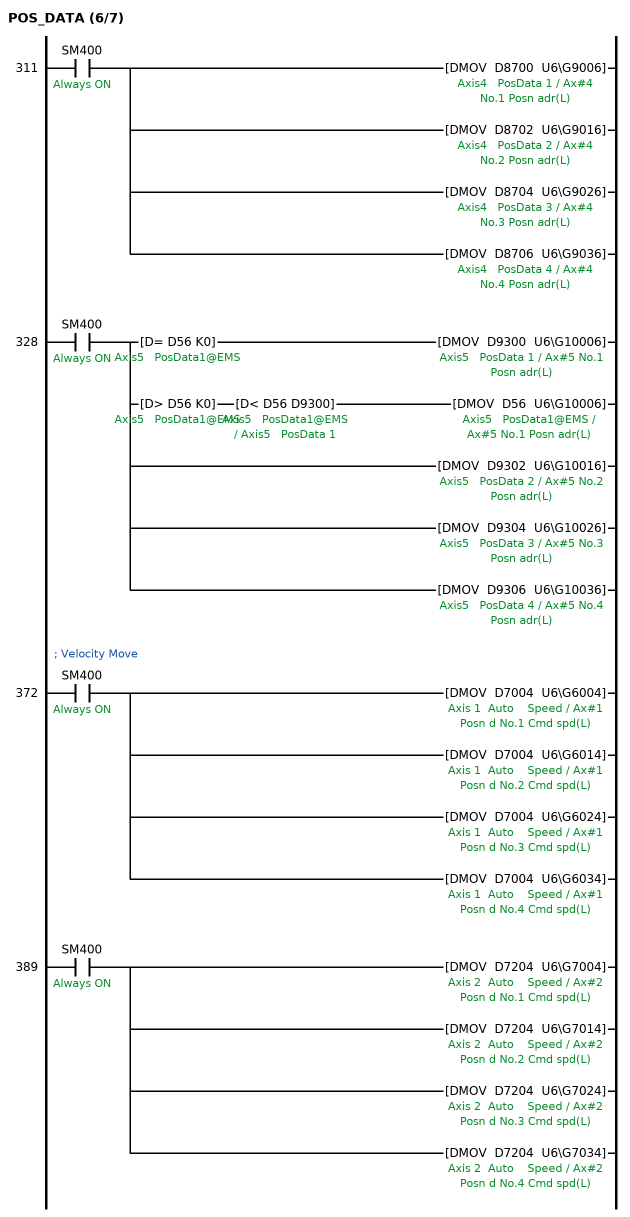
311   LD      SM400  ; Always ON
      DMOV    D8700 U6\G9006  ; Ax#4 No.1 Posn adr(L)
      DMOV    D8702 U6\G9016  ; Ax#4 No.2 Posn adr(L)
      DMOV    D8704 U6\G9026  ; Ax#4 No.3 Posn adr(L)
      DMOV    D8706 U6\G9036  ; Ax#4 No.4 Posn adr(L)
328   LD      SM400  ; Always ON
      MPS
      ANDD=   D56 K0  ; Axis5   PosData1@EMS
      DMOV    D9300 U6\G10006  ; Ax#5 No.1 Posn adr(L)
      MRD
      ANDD>   D56 K0  ; Axis5   PosData1@EMS
      ANDD<   D56 D9300  ; Axis5   PosData1@EMS / Axis5   PosData 1
      DMOV    D56 U6\G10006
      MPP
      DMOV    D9302 U6\G10016  ; Ax#5 No.2 Posn adr(L)
      DMOV    D9304 U6\G10026  ; Ax#5 No.3 Posn adr(L)
      DMOV    D9306 U6\G10036  ; Ax#5 No.4 Posn adr(L)
; Velocity Move
372   LD      SM400  ; Always ON
      DMOV    D7004 U6\G6004  ; Axis 1  Auto    Speed / Ax#1 Posn d No.1 Cmd spd(L)
      DMOV    D7004 U6\G6014  ; Ax#1 Posn d No.2 Cmd spd(L)
      DMOV    D7004 U6\G6024  ; Ax#1 Posn d No.3 Cmd spd(L)
      DMOV    D7004 U6\G6034  ; Ax#1 Posn d No.4 Cmd spd(L)
389   LD      SM400  ; Always ON
      DMOV    D7204 U6\G7004  ; Axis 2  Auto    Speed / Ax#2 Posn d No.1 Cmd spd(L)
      DMOV    D7204 U6\G7014  ; Ax#2 Posn d No.2 Cmd spd(L)
      DMOV    D7204 U6\G7024  ; Ax#2 Posn d No.3 Cmd spd(L)
      DMOV    D7204 U6\G7034  ; Ax#2 Posn d No.4 Cmd spd(L)
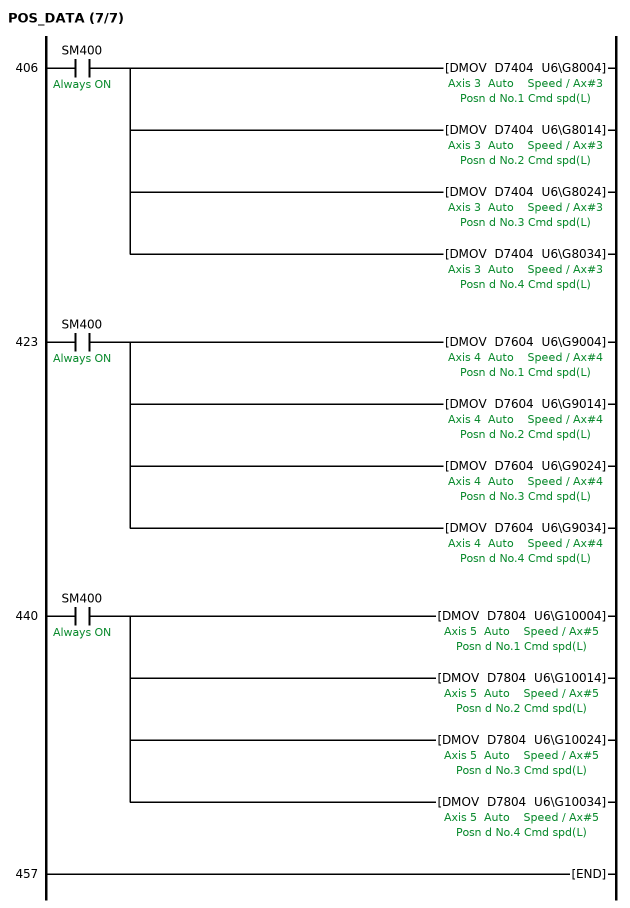
406   LD      SM400  ; Always ON
      DMOV    D7404 U6\G8004  ; Axis 3  Auto    Speed / Ax#3 Posn d No.1 Cmd spd(L)
      DMOV    D7404 U6\G8014  ; Ax#3 Posn d No.2 Cmd spd(L)
      DMOV    D7404 U6\G8024  ; Ax#3 Posn d No.3 Cmd spd(L)
      DMOV    D7404 U6\G8034  ; Ax#3 Posn d No.4 Cmd spd(L)
423   LD      SM400  ; Always ON
      DMOV    D7604 U6\G9004  ; Axis 4  Auto    Speed / Ax#4 Posn d No.1 Cmd spd(L)
      DMOV    D7604 U6\G9014  ; Ax#4 Posn d No.2 Cmd spd(L)
      DMOV    D7604 U6\G9024  ; Ax#4 Posn d No.3 Cmd spd(L)
      DMOV    D7604 U6\G9034  ; Ax#4 Posn d No.4 Cmd spd(L)
440   LD      SM400  ; Always ON
      DMOV    D7804 U6\G10004  ; Axis 5  Auto    Speed / Ax#5 Posn d No.1 Cmd spd(L)
      DMOV    D7804 U6\G10014  ; Ax#5 Posn d No.2 Cmd spd(L)
      DMOV    D7804 U6\G10024  ; Ax#5 Posn d No.3 Cmd spd(L)
      DMOV    D7804 U6\G10034  ; Ax#5 Posn d No.4 Cmd spd(L)
457   END
END_PROGRAM

PROGRAM PB
0     END
END_PROGRAM

// device comments not shown above
M20  ; Manual/ Auto    Select
M996  ; C/V     Auto    Test    Off
M1701  ; Model   No.1
M1702  ; Model   No.2
M1703  ; Model   No.3
M1704  ; Model   No.4
M1705  ; Model   No.5
M1706  ; Model   No.6
M1707  ; Model   No.7
M1708  ; Model   No.8
M1709  ; Model   No.9
M1710  ; Model   No.10
M2010  ; A/M 1   Wait    Vision  Product
M2642  ; C/V 9
M2646  ; C/V 10
M2650  ; C/V 11
M3522  ; Axis5   Offset  Pos     Move
M3552  ; Axis5   Move    2nd Pos Manual
M3566  ; Axis5   Move    Jog+    More
M3568  ; Axis5   Move    Manual  Step4
M3820  ; Vision  Check & delay
M4042  ; O/M 7   Slate   CV      Origin
M6022  ; Tact    Time    Restart 2
Y75  ; Ax#6 Positioning start
Y76  ; Ax#7 Positioning start
Y77  ; Ax#8 Positioning start
Y78  ; Ax#9 Positioning start
Y79  ; Ax#10 Positioning start
Y7A  ; Ax#11 Positioning start
Y7B  ; Ax#12 Positioning start
Y7C  ; Ax#13 Positioning start
Y7D  ; Ax#14 Positioning start
Y7E  ; Ax#15 Positioning start
Y7F  ; Ax#16 Positioning start
Y224  ; PunchingFWD-1
Y225  ; PunchingREV-1
Y226  ; PunchingFWD-2
Y227  ; PunchingREV-2
Y228  ; PunchingFWD-3
Y229  ; PunchingREV-3
Y22A  ; Burring FWD-1
Y22B  ; Burring REV-1
Y22C  ; Burring FWD-2
Y22D  ; Burring REV-2
Y22E  ; Burring FWD-3
Y22F  ; Burring REV-3
Y23A  ; PunchingCLAMP
Y23B  ; PunchingUnCLAMP
Y23C  ; Burring CLAMP
Y23D  ; Burring UnCLAMP
X0A  ; Vision Trigger On Ack
X2C  ; Transfer Jig    Check 1
X2D  ; Transfer Jig    Check 2
X2F  ; Transfer Product Check 1
X33  ; Signal  From TS
X61  ; Synchronization flag
X75  ; Axis #6 BUSY
X76  ; Axis #7 BUSY
X77  ; Axis #8 BUSY
X78  ; Axis #9 BUSY
X79  ; Axis #10 BUSY
X7A  ; Axis #11 BUSY
X7B  ; Axis #12 BUSY
X7C  ; Axis #13 BUSY
X7D  ; Axis #14 BUSY
X7E  ; Axis #15 BUSY
X7F  ; Axis #16 BUSY
X200  ; PunchingFWD-1   Px
X201  ; PunchingREV-1   Px
X202  ; PunchingFWD-2   Px
X203  ; PunchingREV-2   Px
X204  ; PunchingFWD-3   Px
X205  ; PunchingREV-3   Px
X206  ; PunchingCHECK   P/H
X207  ; PunchingUnCLAMP Px
X208  ; Burring FWD-1   Px
X209  ; Burring REV-1   Px
X20A  ; Burring FWD-2   Px
X20B  ; Burring REV-2   Px
X20C  ; Burring FWD-3   Px
X20D  ; Burring REV-3   Px
X20E  ; Burring CHECK   P/H
X20F  ; Burring UnCLAMP  Px
X210  ; 펀칭 양수 1
X211  ; 버링 양수 1
X212  ; 펀칭 양수 2
X213  ; 버링 양수 2
X214  ; PunchingCLAMP   Px
X215  ; Burring CLAMP    Px
X216  ; Spider  Check
X217  ; 유압체크
X21C  ; 펀칭 비상정지
X21D  ; 퍼칭 리셋
X21E  ; 버링 비상정지
X21F  ; 버링 리셋
D4120  ; TP      System  Start   Address
D4300  ; TP      WatchdogWrite   Address
T210  ; A/M 1   Wait    Vision  Product
T363  ; Axis5   Home    Comp    DT@Home
T395  ; Y이동
T432  ; Encoder Unit    Origin  OffDelay
T542  ; C/V 9
T546  ; C/V 10
T550  ; C/V 11
T800  ; Vision  Check & delay
T902  ; 펀칭 양수 딜레이 1
T904  ; 펀칭 Clamp On
T906  ; 펀칭 시작
T908  ; 펀칭 완료 후 펀칭 후진
T910  ; 펀칭후진 완료 후 Clamp 후진
T912  ; 펀칭완료
T952  ; 버링 양수 딜레이 1
T954  ; 버링 Clamp On
T956  ; 버링 시작
T958  ; 버링완료 후 버링 후진
T960  ; 버링후진 완료 후 Clamp 후진
T962  ; 버링완료
W100A  ; Axis6   Current Position
W100C  ; Axis7   Current Position
W100E  ; Axis8   Current Position
W1010  ; Axis9   Current Position
W1012  ; Axis10  Current Position
W1014  ; Axis11  Current Position
W1016  ; Axis12  Current Position
W1018  ; Axis13  Current Position
W101A  ; Axis14  Current Position
W101C  ; Axis15  Current Position
W101E  ; Axis16  Current Position
W1100  ; Axis1   Feedrate
W1102  ; Axis2   Feedrate
W1104  ; Axis3   Feedrate
W1106  ; Axis4   Feedrate
W1108  ; Axis5   Feedrate
W110A  ; Axis6   Feedrate
W110C  ; Axis7   Feedrate
W110E  ; Axis8   Feedrate
W1110  ; Axis9   Feedrate
W1112  ; Axis10  Feedrate
W1114  ; Axis11  Feedrate
W1116  ; Axis12  Feedrate
W1118  ; Axis13  Feedrate
W111A  ; Axis14  Feedrate
W111C  ; Axis15  Feedrate
W111E  ; Axis16  Feedrate
W1205  ; Axis6   Error
W1206  ; Axis7   Error
W1207  ; Axis8   Error
W1208  ; Axis9   Error
W1209  ; Axis10  Error
W120A  ; Axis11  Error
W120B  ; Axis12  Error
W120C  ; Axis13  Error
W120D  ; Axis14  Error
W120E  ; Axis15  Error
W120F  ; Axis16  Error
W1300  ; Axis1   Eff     Load
W1302  ; Axis2   Eff     Load
W1304  ; Axis3   Eff     Load
W1306  ; Axis4   Eff     Load
W1308  ; Axis5   Eff     Load
W130A  ; Axis6   Eff     Load
W130C  ; Axis7   Eff     Load
W130E  ; Axis8   Eff     Load
W1310  ; Axis9   Eff     Load
W1312  ; Axis10  Eff     Load
W1314  ; Axis11  Eff     Load
W1316  ; Axis12  Eff     Load
W1318  ; Axis13  Eff     Load
W131A  ; Axis14  Eff     Load
W131C  ; Axis15  Eff     Load
W131E  ; Axis16  Eff     Load
W1400  ; Axis1   Regen   Load    Ratio
W1401  ; Axis2   Regen   Load    Ratio
W1402  ; Axis3   Regen   Load    Ratio
W1403  ; Axis4   Regen   Load    Ratio
W1404  ; Axis5   Regen   Load    Ratio
W1405  ; Axis6   Regen   Load    Ratio
W1406  ; Axis7   Regen   Load    Ratio
W1407  ; Axis8   Regen   Load    Ratio
W1408  ; Axis9   Regen   Load    Ratio
W1409  ; Axis10  Regen   Load    Ratio
W140A  ; Axis11  Regen   Load    Ratio
W140B  ; Axis12  Regen   Load    Ratio
W140C  ; Axis13  Regen   Load    Ratio
W140D  ; Axis14  Regen   Load    Ratio
W140E  ; Axis15  Regen   Load    Ratio
W140F  ; Axis16  Regen   Load    Ratio
W1500  ; Axis1   Axis    Oper    Status
W1501  ; Axis2   Axis    Oper    Status
W1502  ; Axis3   Axis    Oper    Status
W1503  ; Axis4   Axis    Oper    Status
W1504  ; Axis5   Axis    Oper    Status
W1505  ; Axis6   Axis    Oper    Status
W1506  ; Axis7   Axis    Oper    Status
W1507  ; Axis8   Axis    Oper    Status
W1508  ; Axis9   Axis    Oper    Status
W1509  ; Axis10  Axis    Oper    Status
W150A  ; Axis11  Axis    Oper    Status
W150B  ; Axis12  Axis    Oper    Status
W150C  ; Axis13  Axis    Oper    Status
W150D  ; Axis14  Axis    Oper    Status
W150E  ; Axis15  Axis    Oper    Status
W150F  ; Axis16  Axis    Oper    Status
W1600  ; Axis1   Ext     Input   Sig
W1601  ; Axis2   Ext     Input   Sig
W1602  ; Axis3   Ext     Input   Sig
W1603  ; Axis4   Ext     Input   Sig
W1604  ; Axis5   Ext     Input   Sig
W1605  ; Axis6   Ext     Input   Sig
W1606  ; Axis7   Ext     Input   Sig
W1607  ; Axis8   Ext     Input   Sig
W1608  ; Axis9   Ext     Input   Sig
W1609  ; Axis10  Ext     Input   Sig
W160A  ; Axis11  Ext     Input   Sig
W160B  ; Axis12  Ext     Input   Sig
W160C  ; Axis13  Ext     Input   Sig
W160D  ; Axis14  Ext     Input   Sig
W160E  ; Axis15  Ext     Input   Sig
W160F  ; Axis16  Ext     Input   Sig
W1700  ; Axis1   Status
W1701  ; Axis2   Status
W1702  ; Axis3   Status
W1703  ; Axis4   Status
W1704  ; Axis5   Status
W1705  ; Axis6   Status
W1706  ; Axis7   Status
W1707  ; Axis8   Status
W1708  ; Axis9   Status
W1709  ; Axis10  Status
W170A  ; Axis11  Status
W170B  ; Axis12  Status
W170C  ; Axis13  Status
W170D  ; Axis14  Status
W170E  ; Axis15  Status
W170F  ; Axis16  Status
W1B05  ; Axis6   Warning
W1B06  ; Axis7   Warning
W1B07  ; Axis8   Warning
W1B08  ; Axis9   Warning
W1B09  ; Axis10  Warning
W1B0A  ; Axis11  Warning
W1B0B  ; Axis12  Warning
W1B0C  ; Axis13  Warning
W1B0D  ; Axis14  Warning
W1B0E  ; Axis15  Warning
W1B0F  ; Axis16  Warning
W1705.4  ; Axis6   Org Ok
W1706.4  ; Axis7   Org Ok
W1707.4  ; Axis8   Org Ok
W1708.4  ; Axis9   Org Ok
W1709.4  ; Axis10  Org Ok
W170A.4  ; Axis11  Org Ok
W170B.4  ; Axis12  Org Ok
W170C.4  ; Axis13  Org Ok
W170D.4  ; Axis14  Org Ok
W170E.4  ; Axis15  Org Ok
W170F.4  ; Axis16  Org Ok
D8900.4  ; Vision Change
